TYPE EN_SequenceStartNames :
(
	SequenceStartNamesStart:=10,
	SequenceStartNamesWait:=100,
	SequenceStartNamesDone:=200,
	SequenceStartNamesInit:=300,
	SequenceStartNamesStop:=400
);
END_TYPE

(* stored: Version 1.1.0.1, ProductVersion 3.1.0.36
   DUT EN_SequenceStartNames: Id {822054e7-65a4-4fd5-9889-5b4e32623f94} *)
